# EPICS autosave request: soft_iocs/meas_comp_etc/iocBoot/iocmeas_comp_etc/auto_settings.req
file "ETC_settings.req", P=18ID:ETC:
